{attribute 'qualified_only'}
{attribute 'strict'}
TYPE E_StateSeparatingAutoClamp :
(
	Init 			:= 0,
	Start,
	CloseClamp,
	OpenBarrier,
	CloseBarrier,
	OpenClamp
);
END_TYPE

(* stored: Version 1.1.0.1, ProductVersion 3.1.4024.15
   DUT E_StateSeparatingAutoClamp: Id {3bb431fc-d0a7-4269-85fa-ef5d2aa1e043} *)
